PROGRAM PRG_TXI_VAC_VALVES
VAR

END_VAR

END_PROGRAM

(* stored: Version 1.1.0.1, ProductVersion 3.1.4024.6
   POU PRG_TXI_VAC_VALVES: Id {e927dcd4-ebf1-4ef3-837f-3b457a096b9c}, SpecialFunc None *)
